// TIA Portal V21 export
TYPE "Std_Sequenza"
   STRUCT
      Prm : Struct
         Passo : Array[0.."K_NumPassi"] of Struct
            Durata { S7_SetPoint := 'True'} : "Std_stTimer";
         END_STRUCT;
      END_STRUCT;
      Hmi : Struct
         Stato : Int;   // 1=Ferma 2=InCorso
         BloccaAvanzamento : Bool;   // Impedisce al passo di andare allo stato successivo
         ArrestaSequenza : Bool;   // Riporta la sequenza nel passo zero
         AvviaSequenza : Bool;   // Porta la sequenza nel passo 1
         AvviaSequenzaDisabilitato : Bool;   // Abilitazione a far partire la sequenza
         TempoRimanente : Real;   // Espresso in minuti
         SaltaPasso : Struct   // Funzione che, se abilitata permette all'operatore di skippare determinate condizioni nel passo
            Abilitato : Bool;   // Abilitazione della funzione per operatore
            Richiesto : Bool;   // Richiesta dell'operatore di skippare le condizioni del passo attuale
         END_STRUCT;
         AttendiAckOpertore : Struct   // Funzione che prima di passare al passo successivo richiede una conferma ad HMI dell'operatore
            AbilitaFunz : Bool;   // Abilitazione della funzione per operatore
            AckOperatore : Bool;   // Conferma dell'operatore di passare al passo successivo
         END_STRUCT;
         Diagnostica : Struct   // Funzione utile all'operatore per sapere cosa manca al passo per andare allo stato successivo
            AttesaValvola : Int;   // Attesa della valvola nella posizione richiesta
            AttesaMotore : Int;   // Attesa del motore nello stato corretto
            AttesaAnalogica : Int;   // Attesa dell'analogica nello stato corretto
            AttesaPortata : Int;   // Attesa della portata nello stato corretto
            AttesaExtCondi : Bool;   // Attesa del consenso esterno (condizioni esterne)
            AttesaTempo : Bool;   // Attesa del tempo del passo i corso
            PassoNonAbilitato : Bool;   // Verificare condizioni di abilitazione passo
         END_STRUCT;
      END_STRUCT;
      Dati : Struct
         PassoAttuale : Int;
         TutteLeUtenzeInPosizione : Bool;
         AbilitazionePasso : Bool;
         TempoRimanente : Real;
         TempoTerminato_AttesaCondExt : Bool;
         ResettaTuttiFlipFlop : Bool;   // Necessaria tra una fase e l'altra per essere sicuri che i flip flop siano resettati
         MemoPassoAttuale : Int;
         PrimoGiroPasso : Bool;
      END_STRUCT;
      Allarmi : Struct   // Allarmi Attivi
         "A" : Array[0.."K_NumAllarmiPerSequenza"] of "Std_PrmAllarmeStd";
         WordHMI : Word;   // Word per lista segnalazioni HMI
      END_STRUCT;
      Out : Struct
         SequenzaAvviata : Bool;
         Passo : Array[0.."K_NumPassi"] of Struct
            Attivo { S7_SetPoint := 'True'} : Bool;
         END_STRUCT;
      END_STRUCT;
   END_STRUCT;
END_TYPE
